{attribute 'qualified_only'}
{attribute 'strict'}
TYPE Devices_Secure :
(
	VacuumGripper_MS := 0,
	VacuumGripper_C
);
END_TYPE

(* stored: Version 1.1.0.1, ProductVersion 3.1.4022.12
   DUT Devices_Secure: Id {64f6473d-7818-4e5d-982b-e614ffff07cf} *)
